Xinje XDPPro project, PLC1: XD5-48T6 (software 3.5.3 2018-11-19)

PROGRAM Ladder

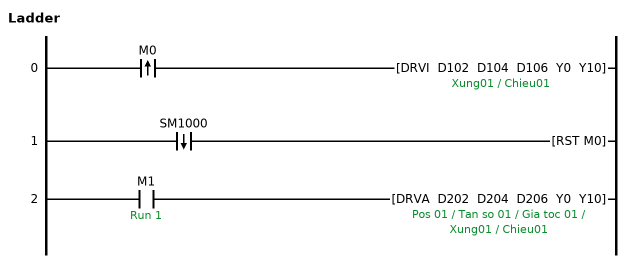
LDP    M0
DRVI   D102 D104 D106 Y0 Y10	; Xung01 / Chieu01
LDF    SM1000
RST    M0
LD     M1	; Run 1
DRVA   D202 D204 D206 Y0 Y10	; Pos 01 / Tan so 01 / Gia toc 01 / Xung01 / Chieu01

COMMENTS (devices not used above)
Y7	Chieu01